FUNCTION_BLOCK AX_XOR_3_UNGATED (* FB to calculate boolean XOR (generic FB) OHNE Aenderungserkennung - reicht JEDES neu berechnete Ergebnis bedingungslos weiter (fuer Verbraucher, die eine periodische Kadenz unabhaengig von Wertaenderung brauchen, z.B. Ableitungs-/Frequenzberechnungen). *)
  (* Standard: 61499-2; Description: Copyright (c) 2026 Meisterschulen am Ostbahnhof This program and the accompanying materials are made available under the terms of the Eclipse Public License 2.0 which is available at https://www.eclipse.org/legal/epl-2.0/ SPDX-License-Identifier: EPL-2.0 *)
  (* Version 1.0, 2026-08-31, Franz Höpfinger, HR Agrartechnik GmbH *)
  PACKAGE adapter::booleanOperators;
  IMPORT eclipse4diac::core::GenericClassName;
  {SET_ATTRIBUTE(eclipse4diac::core::GenericClassName, 'GEN_AX_XOR')}
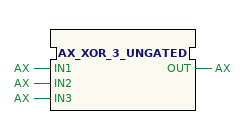
  SOCKETS
    IN1 : adapter::types::unidirectional::AX; (* XOR input 1 *)
    IN2 : adapter::types::unidirectional::AX; (* XOR input 2 *)
    IN3 : adapter::types::unidirectional::AX; (* XOR input 3 *)
  END_SOCKETS
  PLUGS
    OUT : adapter::types::unidirectional::AX; (* XOR result *)
  END_PLUGS
END_FUNCTION_BLOCK
